ABB RAPID module: MainModule.mod

MODULE MainModule
LOCAL CONST string YuMi_App_Program_Version:="1.0.1"; !Do not edit or remove this line!
LOCAL VAR robtarget s43 := [[416.87,26.87,105.67],[0.239717,0.600269,0.690366,0.324974],[-2,2,0,11],[129.868,9E+09,9E+09,9E+09,9E+09,9E+09]];
LOCAL VAR robtarget s42 := [[382.53,-123.02,10.53],[0.244689,0.674836,0.65128,0.246086],[-2,2,0,11],[141.993,9E+09,9E+09,9E+09,9E+09,9E+09]];
LOCAL VAR robtarget s41 := [[425.29,-119.25,-11.96],[0.259693,0.659374,0.65786,0.254962],[-2,2,0,11],[136.632,9E+09,9E+09,9E+09,9E+09,9E+09]];
LOCAL VAR robtarget s40 := [[425.28,-119.78,-6.33],[0.253223,0.670513,0.653273,0.243977],[-2,2,0,11],[135.935,9E+09,9E+09,9E+09,9E+09,9E+09]];
LOCAL VAR robtarget s39 := [[404.49,-110.47,21.27],[0.373447,0.638614,0.631836,0.231285],[-2,2,0,11],[132.435,9E+09,9E+09,9E+09,9E+09,9E+09]];
LOCAL VAR robtarget s38 := [[366.21,-90.09,26.98],[0.335027,-0.242508,0.901449,-0.127812],[-2,2,-1,11],[123.264,9E+09,9E+09,9E+09,9E+09,9E+09]];
LOCAL VAR robtarget s37 := [[522.17,124.54,100.86],[0.27966,0.555394,0.695933,0.359172],[-2,2,0,11],[126.812,9E+09,9E+09,9E+09,9E+09,9E+09]];
LOCAL VAR robtarget s36 := [[386.85,-114.71,20.70],[0.264578,0.652526,0.671108,0.231998],[-2,2,0,11],[130.466,9E+09,9E+09,9E+09,9E+09,9E+09]];
LOCAL VAR robtarget s35 := [[425.42,-118.22,-11.79],[0.263538,0.648196,0.671667,0.24342],[-2,2,0,11],[125.698,9E+09,9E+09,9E+09,9E+09,9E+09]];
LOCAL VAR robtarget s34 := [[408.83,-115.82,1.80],[0.255631,0.654448,0.654837,0.278459],[-2,2,0,11],[126.406,9E+09,9E+09,9E+09,9E+09,9E+09]];
LOCAL VAR robtarget s33 := [[376.14,-84.73,20.05],[0.267639,0.336867,0.892346,0.136412],[-2,2,-1,11],[122.413,9E+09,9E+09,9E+09,9E+09,9E+09]];
LOCAL VAR robtarget s32 := [[418.24,-45.52,-18.61],[0.14668,-0.836617,0.421461,-0.317692],[-2,2,-2,11],[117.09,9E+09,9E+09,9E+09,9E+09,9E+09]];
LOCAL VAR robtarget s31 := [[486.79,17.58,-17.97],[0.289285,-0.684492,0.611031,-0.272811],[-2,2,-2,11],[121.251,9E+09,9E+09,9E+09,9E+09,9E+09]];
LOCAL VAR robtarget s30 := [[486.79,17.58,-17.98],[0.289284,-0.684495,0.611031,-0.272804],[-2,2,-2,11],[121.251,9E+09,9E+09,9E+09,9E+09,9E+09]];
LOCAL VAR robtarget s29 := [[497.61,52.17,25.68],[0.0744218,0.982371,-0.133398,-0.107762],[-2,0,-3,11],[-144.393,9E+09,9E+09,9E+09,9E+09,9E+09]];
LOCAL VAR robtarget s28 := [[498.96,-106.34,12.85],[0.154271,0.656781,-0.720962,-0.158283],[-2,0,-2,11],[-127.622,9E+09,9E+09,9E+09,9E+09,9E+09]];
LOCAL VAR robtarget s27 := [[446.14,-112.43,-11.49],[0.231446,0.679733,-0.660009,-0.220873],[-2,0,-2,11],[-74.4768,9E+09,9E+09,9E+09,9E+09,9E+09]];
LOCAL VAR robtarget s26 := [[464.77,-112.97,-6.12],[0.209965,0.687195,-0.664398,-0.205556],[-2,1,-2,11],[-101.314,9E+09,9E+09,9E+09,9E+09,9E+09]];
LOCAL VAR robtarget s25 := [[469.07,-108.51,1.73],[0.2009,0.692042,-0.657786,-0.219167],[-2,1,-2,11],[-101.923,9E+09,9E+09,9E+09,9E+09,9E+09]];
LOCAL VAR robtarget s24 := [[454.79,-115.80,-5.05],[0.22027,0.661073,-0.684542,-0.214163],[-2,1,-2,11],[150.757,9E+09,9E+09,9E+09,9E+09,9E+09]];
LOCAL VAR robtarget s23 := [[501.20,-61.57,54.22],[0.1235,0.756883,-0.639624,-0.0525036],[-2,1,-2,11],[125.887,9E+09,9E+09,9E+09,9E+09,9E+09]];
LOCAL VAR robtarget s22 := [[519.03,5.74,27.98],[0.277262,-0.737207,0.474269,-0.393345],[-2,2,-2,11],[118.466,9E+09,9E+09,9E+09,9E+09,9E+09]];
LOCAL VAR robtarget s21 := [[461.58,12.19,-82.83],[0.309126,-0.642585,0.641597,-0.282626],[-2,2,-2,11],[124.855,9E+09,9E+09,9E+09,9E+09,9E+09]];
LOCAL VAR robtarget s20 := [[465.21,15.46,30.59],[0.0721419,0.732955,-0.676317,-0.0129994],[-2,1,-2,11],[132.33,9E+09,9E+09,9E+09,9E+09,9E+09]];
LOCAL VAR robtarget s19 := [[507.00,-11.26,3.56],[0.350028,-0.617528,0.59609,-0.375255],[-2,2,-2,11],[121.613,9E+09,9E+09,9E+09,9E+09,9E+09]];
LOCAL VAR robtarget s18 := [[460.68,10.06,-85.04],[0.303428,-0.647195,0.64014,-0.281586],[-2,2,-2,11],[124.868,9E+09,9E+09,9E+09,9E+09,9E+09]];
LOCAL VAR robtarget s17 := [[461.59,12.21,-82.83],[0.309165,-0.64258,0.641584,-0.282627],[-2,2,-2,11],[124.853,9E+09,9E+09,9E+09,9E+09,9E+09]];
LOCAL VAR robtarget s16 := [[463.29,-0.43,-24.31],[0.0442281,0.694541,-0.711551,-0.0967084],[-2,1,-2,11],[117.142,9E+09,9E+09,9E+09,9E+09,9E+09]];
LOCAL VAR robtarget s15 := [[465.73,9.70,-2.98],[0.328984,-0.660159,0.614742,-0.279379],[-2,2,-2,11],[115.561,9E+09,9E+09,9E+09,9E+09,9E+09]];
LOCAL VAR robtarget s14 := [[443.70,-124.14,-5.18],[0.310242,-0.657967,0.589823,-0.350626],[-2,2,-2,11],[122.972,9E+09,9E+09,9E+09,9E+09,9E+09]];
LOCAL VAR robtarget s13 := [[408.55,-120.12,-61.99],[0.280554,-0.661564,0.63124,-0.291819],[-2,2,-2,11],[126.614,9E+09,9E+09,9E+09,9E+09,9E+09]];
LOCAL VAR robtarget s12 := [[406.34,-119.87,-55.26],[0.308534,-0.6582,0.610035,-0.315336],[-2,2,-2,11],[123.638,9E+09,9E+09,9E+09,9E+09,9E+09]];
LOCAL VAR robtarget s11 := [[417.82,-90.47,-11.35],[0.206194,-0.582261,0.722747,-0.30999],[-2,2,-2,11],[118.803,9E+09,9E+09,9E+09,9E+09,9E+09]];
LOCAL VAR robtarget s10 := [[485.54,-36.45,-28.70],[0.00698082,0.286245,-0.955057,0.0766916],[-2,1,-1,11],[127.675,9E+09,9E+09,9E+09,9E+09,9E+09]];
LOCAL VAR robtarget s9 := [[481.71,-54.99,-68.15],[0.00986987,-0.271898,0.957628,-0.0944646],[-2,1,-1,11],[130.998,9E+09,9E+09,9E+09,9E+09,9E+09]];
LOCAL VAR robtarget s8 := [[407.82,-120.06,-62.23],[0.299734,-0.651529,0.626303,-0.305636],[-2,2,-2,11],[131.051,9E+09,9E+09,9E+09,9E+09,9E+09]];
LOCAL VAR robtarget s7 := [[408.15,-120.93,-53.24],[0.300014,-0.650343,0.633333,-0.293145],[-2,2,-2,11],[130.944,9E+09,9E+09,9E+09,9E+09,9E+09]];
LOCAL VAR robtarget s6 := [[404.26,-93.36,-10.76],[0.304779,-0.648376,0.61805,-0.323624],[-2,2,-2,11],[127.666,9E+09,9E+09,9E+09,9E+09,9E+09]];
LOCAL VAR robtarget s5 := [[490.69,-26.58,-4.99],[0.0269535,0.170548,-0.983687,0.0504678],[-2,1,-1,11],[123.39,9E+09,9E+09,9E+09,9E+09,9E+09]];
LOCAL VAR robtarget s4 := [[481.57,-55.15,-68.21],[0.0106894,-0.27072,0.958035,-0.0936206],[-2,1,-1,11],[131.076,9E+09,9E+09,9E+09,9E+09,9E+09]];
LOCAL VAR robtarget s3 := [[479.76,-48.95,-56.71],[0.0161053,-0.263449,0.956876,-0.121344],[-2,1,-1,11],[129.594,9E+09,9E+09,9E+09,9E+09,9E+09]];
LOCAL VAR robtarget s2 := [[456.48,5.63,28.15],[0.0713279,-0.283227,0.854876,-0.428814],[-2,1,-1,11],[126.276,9E+09,9E+09,9E+09,9E+09,9E+09]];
LOCAL VAR robtarget s1 := [[358.37,68.26,133.15],[0.275359,-0.042554,0.863052,-0.421316],[-1,1,0,11],[117.323,9E+09,9E+09,9E+09,9E+09,9E+09]];
PROC main()
MoveSync s1;
MoveSync s2;
MoveSync s3;
MoveSync s9;
CloseHand;
MoveSync s10;
MoveSync s11;
MoveSync s12;
MoveSync s13;
OpenHand;
MoveSync s14;
MoveSync s15;
MoveSync s17;
CloseHand;
MoveSync s30;
MoveSync s31;
MoveSync s32;
MoveSync s38;
MoveSync s39;
MoveSync s40;
MoveSync s41;
OpenHand;
MoveSync s42;
MoveSync s43;
ENDPROC
ENDMODULE
